	4://区域限定(4:skyRetract)
		CASE phyIdx OF
			0:	lgcIdx := 185;		//sky0r	->	起竖
			1:	lgcIdx := 175;		//sky1r	->	横1
			2:	lgcIdx := 183;		//sky2r	->	纵1
			3:	lgcIdx := 176;		//sky3r	->	横2
			4:	lgcIdx := 177;		//sky4r	->	横3
			5:	lgcIdx := 178;		//sky5r	->	横4
			6:	lgcIdx := 179;		//sky6r	->	横5
			7:	lgcIdx := 184;		//sky7r	->	纵2
			8:	lgcIdx := 180;		//sky8r	->	横6
			9:	lgcIdx := 181;		//sky9r	->	横7
			10:	lgcIdx := 182;		//sky10r->	横8
		END_CASE
END_CASE

END_FUNCTION_BLOCK

// Device/Application/modbus/mdbsNumToIdx
FUNCTION_BLOCK mdbsNumToIdx
VAR_INPUT
	devNo		:WORD;
END_VAR
VAR_OUTPUT
	level		:INT;
	idx			:INT;
END_VAR
VAR
	
END_VAR

IF devNo > 40000 THEN
	CASE devNo OF
		//地轨
		41010:	level := 1;	idx := 1;
		41020:	level := 1;	idx := 3;
		41030:	level := 1;	idx := 4;
		41040:	level := 1;	idx := 5;
		41050:	level := 1;	idx := 6;
		41060:	level := 1;	idx := 8;
		41070:	level := 1;	idx := 9;
		41080:	level := 1;	idx := 10;
		42010:	level := 1;	idx := 2;
		42020:	level := 1;	idx := 7;
		
		51010:	level := 2;	idx := 1;
		51020:	level := 2;	idx := 3;
		51030:	level := 2;	idx := 4;
		51040:	level := 2;	idx := 5;
		51050:	level := 2;	idx := 6;
		51060:	level := 2;	idx := 8;
		51070:	level := 2;	idx := 9;
		51080:	level := 2;	idx := 10;
		52010:	level := 2;	idx := 2;
		52020:	level := 2;	idx := 7;
		53000:	level := 2;	idx := 0;
		53010:	level := 2;	idx := 0;
	END_CASE
END_IF

END_FUNCTION_BLOCK

// Device/Application/modbus/DataReverse
FUNCTION_BLOCK DataReverse
VAR_INPUT
END_VAR
VAR_OUTPUT
END_VAR
VAR
END_VAR

METHOD cmdReverse : TargetDirect
VAR_INPUT
	input		:TargetDirect;
END_VAR
IF input = TargetDirect.extend THEN
	cmdReverse := TargetDirect.retract;
END_IF
IF input = TargetDirect.retract THEN
	cmdReverse := TargetDirect.extend;
END_IF
END_METHOD

END_FUNCTION_BLOCK

// Device/Application/healthydata/TcpUploader
PROGRAM TcpUploader
VAR
	destIp 			:STRING:='172.18.150.31';
	destPort 		:UINT:= 61158;
	tcpConnector	:tcpUpload;
	
	myData 			:ARRAY[1..1024]OF BYTE;
	myDataLen		:__XINT:=21 * 3 + 16;		//总数据长度
	
	init			:BOOL :=TRUE;	
END_VAR



//initialize
IF init THEN
	init := FALSE;
	tcpConnector(InetAddress := destIp,port:= destPort);
END_IF

prepareMetaData();

tcpConnector.send(dataLength := myDataLen, sendBuf := myData);

METHOD prepareMetaData
VAR_INPUT
END_VAR
VAR
	gi				:INT;
	si				:INT;
	
	intTmp			:UINT;	
	pos				:INT;
	byte1			:BYTE;
	byte2			:BYTE;
	plugStat		:BYTE;
END_VAR
//data head (decimal)
myData[1]	:=	83	;
myData[2]	:=	70	;
myData[3]	:=	68	;
myData[4]	:=	84	;

//data length
myData[5]	:=	0	;
myData[6]	:=	63	;

//healthy data
myData[7]	:=	0	;
myData[8]	:=	11	;

//zero
myData[9]	:=	0	;
myData[10]	:=	0	;
myData[11]	:=	0	;
myData[12]	:=	0	;

myData[13]	:=	0	;
myData[14]	:=	0	;
myData[15]	:=	0	;
myData[16]	:=	0	;

//list
pos := 17;
FOR gi := 1 TO 10 DO
	intTmp := REAL_TO_UINT(gDev.grd[gi].sensor.position * 10);
	byte1 := UINT_TO_BYTE(SHR(intTmp, 8)); 
	byte2 := UINT_TO_BYTE(intTmp AND 255); 
	plugStat := INT_TO_BYTE(gDev.grd[gi].state);
	
	myData[pos] := plugStat;
	pos := pos + 1;		
	myData[pos] := byte1;
	pos := pos + 1;
	myData[pos] := byte2;
	pos := pos + 1;
END_FOR
FOR si := 0 TO 10 DO
	intTmp := REAL_TO_UINT(gDev.sky[si].sensor.position * 10);
	byte1 := UINT_TO_BYTE(SHR(intTmp, 8)); 
	byte2 := UINT_TO_BYTE(intTmp AND 255); 
	plugStat := INT_TO_BYTE(gDev.sky[si].state);
	
	myData[pos] := plugStat;
	pos := pos + 1;		
	myData[pos] := byte1;
	pos := pos + 1;
	myData[pos] := byte2;
	pos := pos + 1;
END_FOR
END_METHOD

END_PROGRAM

// Device/Application/basefun/tcpUpload
FUNCTION_BLOCK tcpUpload
VAR_INPUT
	InetAddress		:STRING;
	port			:UINT;
END_VAR
VAR_OUTPUT
END_VAR
VAR
	tcpConnector	:TCP.Connector;
	tcpStream		:TCP.Stream;
	pointerStream	:POINTER TO TCP.Stream;


	tcpState		:UINT:=0;
	tcpCount		:UINT:=0;
	
	netState		:INT;


END_VAR

METHOD send
VAR_INPUT
	
	dataLength		:__XINT;
	sendBuf 		:ARRAY[1..1024]OF BYTE;
END_VAR
VAR
	sizeData		:__XINT;
END_VAR

tcpCount := tcpCount + 1;

CASE tcpState OF

	0:			//connet server
		tcpConnector.Connect(sIPAddress:= InetAddress,uiPort:= port,pStream => pointerStream);
		IF pointerStream<>0 THEN
			tcpState :=1;
		ELSE
			tcpState :=2;
		END_IF
		
	1:			
		netState := pointerStream^.Send(ADR(sendBuf),dataLength,diSent=>sizeData);			
		IF netState <> 0 THEN
			tcpState := 2;	
		END_IF
		
		
	2:		 	//断开连接
	    tcpConnector.Disconnect();
		tcpState := 0;

END_CASE
END_METHOD

END_FUNCTION_BLOCK

// Device/Application/healthydata/FileSaver
PROGRAM FileSaver
VAR
	path 			:STRING:='D:/log';
	intervalMs		:INT := 10;		//间隔时间
	
	init			:BOOL:= TRUE;
	gi				:INT;
	si				:INT;	
	cCtrl			:INT;

	sav				:ARRAY[1..2, 0..10] OF fileSave;
	speed			:INT;
	nowCmd			:ARRAY[1..2, 0..10] OF BOOL;
	canWrite		:ARRAY[1..2, 0..10] OF BOOL;
	nowPosition		:ARRAY[1..2, 0..10] OF INT;
	lastPosition	:ARRAY[1..2, 0..10] OF INT;
	state			:ARRAY[1..2, 0..10] OF INT;
	flag			:ARRAY[1..2, 0..10] OF INT;
END_VAR
VAR CONSTANT
	aOil	:ARRAY [1..7] OF INT :=[9,11,8,8,8,8,23];		
END_VAR

//initialize
IF init THEN
	init := FALSE;
	FOR gi := 1 TO 10 DO
		 sav[1, gi](filePath := path, intervalt := intervalMs);
		 sav[1, gi].createDir(gUI.grd[gi].name);
		 init := FALSE;
	END_FOR
	FOR si := 0 TO 10 DO
		 sav[2, si](filePath := path, intervalt := intervalMs);
		 sav[2, si].createDir(gUI.sky[si].name);
		 init := FALSE;
	END_FOR
END_IF

//detect and record ground and sky
FOR gi := 1 TO 10 DO
	 nowCmd[1, gi] := gUI.grd[gi].btnExtend OR gUI.grd[gi].btnRetract;
	 IF nowCmd[1, gi] THEN
		 IF flag[1, gi] = 0 THEN
			 sav[1, gi].new(devName := gUI.grd[gi].name);
			 flag[1, gi] := 1;
		 END_IF
		 //prepare data
		 getGrdData();
		 //write
		 sav[1, gi].write(positionInt := nowPosition[1, gi],speedInt := speed,
			 				 stateInt := state[1, gi]);
	 ELSE
		 IF flag[1, gi] = 1 THEN
			 sav[1, gi].write(positionInt := nowPosition[1, gi],speedInt := speed,
				 				 stateInt := state[1, gi]);
			 sav[1, gi].close();
			 flag[1, gi] := 0;
		 END_IF
	 END_IF
END_FOR


FOR si := 0 TO 10 DO
	 nowCmd[2, si] := gUI.sky[si].btnExtend OR gUI.sky[si].btnRetract;
	 IF nowCmd[2, si] THEN
		 IF flag[2, si] = 0 THEN
			 sav[2, si].new(devName := gUI.sky[si].name);
			 flag[2, si] := 1;
		 END_IF
		 //prepare data
		 getSkyData();
		 //write
		 sav[2, si].write(positionInt := nowPosition[2, si],speedInt := speed,
			 				 stateInt := state[2, si]);
	 ELSE
		 IF flag[2, si] = 1 THEN
			 sav[2, si].write(positionInt := nowPosition[2, si],speedInt := speed,
				 				 stateInt := state[2, si]);
			 sav[2, si].close();
			 flag[2, si] := 0;
		 END_IF
	 END_IF
END_FOR

ACTION getSkyData:
//进制转换 到0.01mm
lastPosition[2, si] := nowPosition[2, si];
nowPosition[2, si] := REAL_TO_INT(10 * gDev.sky[si].sensor.position);

speed := REAL_TO_INT(gDev.sky[si].sensor.speed);


state[2, si] := gDev.sky[si].state;
END_ACTION

ACTION getGrdData:
//进制转换 到0.01mm
lastPosition[1, gi] := nowPosition[1, gi];
nowPosition[1, gi] := REAL_TO_INT(10 * gDev.grd[gi].sensor.position);

speed := REAL_TO_INT(gDev.grd[gi].sensor.speed);


state[1, gi] := gDev.grd[gi].state;
END_ACTION

END_PROGRAM

// Device/Application/basefun/fileSave
FUNCTION_BLOCK fileSave
VAR_INPUT
	filePath 	:STRING;
	intervalt	:INT;
END_VAR
VAR
	lineCount	: INT;
	fileHandle  : DWORD;
	fileName	: STRING;
END_VAR
VAR_OUTPUT
END_VAR

METHOD new

	
VAR_INPUT
	devName		: STRING ;

END_VAR
VAR
	
	fileHandle0 : DWORD;
	datetime	: DATE_AND_TIME;
	UdIntms 	: UDINT;
	UdMsOffset  : UDINT;
	DTimer_Str  : STRING;
	uiYear 		: UINT; 
    uiMonth 	: UINT; 
    uiDay 		: UINT; 
    uiHour 		: UINT; 
    uiMinute 	: UINT; 
    uiSecond 	: UINT;	
	uiMsSecond	: UINT;



	 S_Time64		:  SysTime64;
	 STT			:  CurTimeEx;
	 S_Time			:  SystemTimeDate;
	 Time_Str		:  STRING;
	F_err		: DWORD;
	F_HANDL		: DWORD;

END_VAR

	STT(SystemTime:= S_Time64, TimeDate:= S_Time);
	Time_Str :='';
	Time_Str := concat(Time_Str,UINT_TO_STRING(S_Time.Year));
	Time_Str := concat(Time_Str,'-');
	Time_Str := concat(Time_Str,UINT_TO_STRING(S_Time.Month));
	Time_Str := concat(Time_Str,'-');
	Time_Str := concat(Time_Str,UINT_TO_STRING(S_Time.Day));
	Time_Str := concat(Time_Str,'_');
	Time_Str := concat(Time_Str,UINT_TO_STRING(S_Time.Hour));
	Time_Str := concat(Time_Str,'-');
	Time_Str := concat(Time_Str,UINT_TO_STRING(S_Time.Minute));
	Time_Str := concat(Time_Str,'-');
	Time_Str := concat(Time_Str,UINT_TO_STRING(S_Time.Second));
	Time_Str := concat(Time_Str,'_');
	Time_Str := concat(Time_Str,UINT_TO_STRING(S_Time.Milliseconds));

	fileName := FilePath;
	fileName := concat(fileName,'/');
	fileName := concat(fileName,devName);

	
	fileName := concat(fileName,'/');
	fileName := concat(fileName,devName);
	fileName := concat(fileName,'-');
	fileName := concat(fileName,Time_Str);
    fileName := concat(fileName,'.txt');

	fileHandle := SysFileOpen(szFile:= fileName, am:=ACCESS_MODE.AM_WRITE, pResult:= ADR(F_err));
	lineCount := -1;
	//fileHandle := SysFileOpen(szFile:= fileName, am:=ACCESS_MODE.AM_APPEND, pResult:= ADR(F_err));
END_METHOD

METHOD close
VAR_INPUT
END_VAR
IF fileHandle <> 0 THEN
	SysFileClose(hFile := fileHandle);
	fileHandle := 0;
END_IF
END_METHOD

METHOD write
VAR_INPUT

	positionInt 	:INT;
	speedInt 		:INT;
	stateInt		:INT;
	
END_VAR
VAR
	data		: STRING;
	F_err		: DWORD;
	tempInt		: INT;
END_VAR

IF fileHandle <> 0 THEN
	lineCount := lineCount + 1;
	tempInt	:= lineCount * intervalt;
	data := INT_TO_STRING(lineCount);
	data := concat(data,'$T$T');
	data := concat(data, INT_TO_STRING(tempInt));
	IF tempInt < 1000 THEN
		data := concat(data,'$T');
	END_IF
	data := concat(data,'$T$T');
	data := concat(data,INT_TO_STRING(positionInt));
	data := concat(data,'$T');
	data := concat(data,INT_TO_STRING(speedInt));
	data := concat(data,'$T');
	data := concat(data,INT_TO_STRING(stateInt));
	data := concat(data,'$R');
	
	SysFileWrite(hFile:=fileHandle , pbyBuffer:= ADR(data) , ulSize:= DINT_TO_DWORD(SysStrLen(data)) , pResult:= ADR(F_err));		// 写入数据

END_IF
END_METHOD

METHOD createDir
VAR_INPUT
	devName		: STRING ;
END_VAR
VAR
	filePath1	:STRING;
END_VAR
filePath1 := FilePath;
filePath1 := concat(filePath1,'/');
filePath1 := concat(filePath1,devName);
SysDirCreate2(filePath1, TRUE);
END_METHOD

END_FUNCTION_BLOCK

// Device/Application/visualization/baseModule/DevUnit0
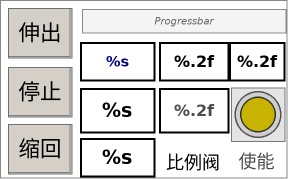
VISUALIZATION DevUnit0  // 288x179
VAR_IN_OUT
	extendButton		: BOOL;
	retractButton		: BOOL;
	stopButton			: BOOL;
	
	percentShow			:REAL;	
	nameShow			:STRING;
	wnameShow			:WSTRING;
	hzname				:WSTRING;
	posShow				:REAL;
	spdShow				:REAL;
	
	pwrEnable			:BOOL;
	pwrPct				:REAL;

END_VAR
    RoundedRectangle (159,88 70x45), "%.2f", text variable: pwrPct
        OnMouseDown: write the text variable via Default, min 0, max 100
    Label (159,149 68x28), "比例阀"
    PushSwitchLed (231,87 54x55), variable: pwrEnable, behaviour: TOGGLE, style: Switch-PushSwitchLed-Yellow
    Label (231,151 51x22), "使能"
    RoundedRectangle (80,42 75x39), "%s", text variable: nameShow
    RoundedRectangle (159,42 70x39), "%.2f", text variable: posShow
    Progressbar (82,9 204x24), variable: percentShow
    Button (8,124 64x50), "缩回"
        toggle retractButton
    Button (8,67 64x50), "停止"
        toggle stopButton
    Button (8,8 64x50), "伸出"
        toggle extendButton
    RoundedRectangle (229,42 56x39), "%.2f", text variable: spdShow
    RoundedRectangle (80,88 75x45), "%s", text variable: wnameShow
    RoundedRectangle (80,138 75x39), "%s", text variable: hzname
END_VISUALIZATION

// Device/Application/visualization/baseModule/grd
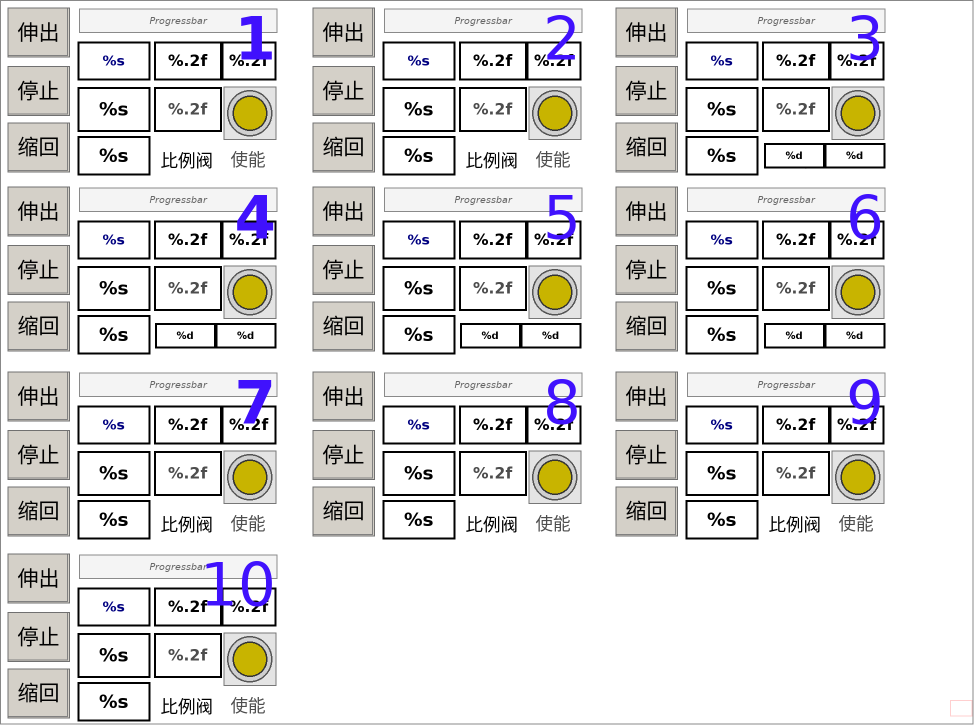
VISUALIZATION grd  // 974x725
    Frame (0,0 279x177), "1"
        shows DevUnit0(extendButton := gUI.grd[1].btnExtend, retractButton := gUI.grd[1].btnRetract, stopButton := gUI.grd[1].btnStop, percentShow := gUI.grd[1].extendPercent, nameShow := gUI.grd[1].name, wnameShow := gUI.grd[1].wname, hzname := gUI.grd[1].hzname, posShow := gUI.grd[1].postion, spdShow := gUI.grd[1].speed, pwrEnable := gUI.grd[1].pwrEnable, pwrPct := gUI.grd[1].pwrPercent)
    Frame (305,0 279x177), "2"
        shows DevUnit0(extendButton := gUI.grd[2].btnExtend, retractButton := gUI.grd[2].btnRetract, stopButton := gUI.grd[2].btnStop, percentShow := gUI.grd[2].extendPercent, nameShow := gUI.grd[2].name, wnameShow := gUI.grd[2].wname, hzname := gUI.grd[2].hzname, posShow := gUI.grd[2].postion, spdShow := gUI.grd[2].speed, pwrEnable := gUI.grd[2].pwrEnable, pwrPct := gUI.grd[2].pwrPercent)
    Frame (608,0 279x177), "3"
        shows DevUnit0(extendButton := gUI.grd[3].btnExtend, retractButton := gUI.grd[3].btnRetract, stopButton := gUI.grd[3].btnStop, percentShow := gUI.grd[3].extendPercent, nameShow := gUI.grd[3].name, wnameShow := gUI.grd[3].wname, hzname := gUI.grd[3].hzname, posShow := gUI.grd[3].postion, spdShow := gUI.grd[3].speed, pwrEnable := gUI.grd[3].pwrEnable, pwrPct := gUI.grd[3].pwrPercent)
    Frame (0,179 279x177), "4"
        shows DevUnit0(extendButton := gUI.grd[4].btnExtend, retractButton := gUI.grd[4].btnRetract, stopButton := gUI.grd[4].btnStop, percentShow := gUI.grd[4].extendPercent, nameShow := gUI.grd[4].name, wnameShow := gUI.grd[4].wname, hzname := gUI.grd[4].hzname, posShow := gUI.grd[4].postion, spdShow := gUI.grd[4].speed, pwrEnable := gUI.grd[4].pwrEnable, pwrPct := gUI.grd[4].pwrPercent)
    Frame (305,179 279x177), "5"
        shows DevUnit0(extendButton := gUI.grd[5].btnExtend, retractButton := gUI.grd[5].btnRetract, stopButton := gUI.grd[5].btnStop, percentShow := gUI.grd[5].extendPercent, nameShow := gUI.grd[5].name, wnameShow := gUI.grd[5].wname, hzname := gUI.grd[5].hzname, posShow := gUI.grd[5].postion, spdShow := gUI.grd[5].speed, pwrEnable := gUI.grd[5].pwrEnable, pwrPct := gUI.grd[5].pwrPercent)
    Frame (608,179 279x177), "6"
        shows DevUnit0(extendButton := gUI.grd[6].btnExtend, retractButton := gUI.grd[6].btnRetract, stopButton := gUI.grd[6].btnStop, percentShow := gUI.grd[6].extendPercent, nameShow := gUI.grd[6].name, wnameShow := gUI.grd[6].wname, hzname := gUI.grd[6].hzname, posShow := gUI.grd[6].postion, spdShow := gUI.grd[6].speed, pwrEnable := gUI.grd[6].pwrEnable, pwrPct := gUI.grd[6].pwrPercent)
    Frame (0,364 279x177), "7"
        shows DevUnit0(extendButton := gUI.grd[7].btnExtend, retractButton := gUI.grd[7].btnRetract, stopButton := gUI.grd[7].btnStop, percentShow := gUI.grd[7].extendPercent, nameShow := gUI.grd[7].name, wnameShow := gUI.grd[7].wname, hzname := gUI.grd[7].hzname, posShow := gUI.grd[7].postion, spdShow := gUI.grd[7].speed, pwrEnable := gUI.grd[7].pwrEnable, pwrPct := gUI.grd[7].pwrPercent)
    Frame (305,364 279x177), "8"
        shows DevUnit0(extendButton := gUI.grd[8].btnExtend, retractButton := gUI.grd[8].btnRetract, stopButton := gUI.grd[8].btnStop, percentShow := gUI.grd[8].extendPercent, nameShow := gUI.grd[8].name, wnameShow := gUI.grd[8].wname, hzname := gUI.grd[8].hzname, posShow := gUI.grd[8].postion, spdShow := gUI.grd[8].speed, pwrEnable := gUI.grd[8].pwrEnable, pwrPct := gUI.grd[8].pwrPercent)
    Frame (608,364 279x177), "9"
        shows DevUnit0(extendButton := gUI.grd[9].btnExtend, retractButton := gUI.grd[9].btnRetract, stopButton := gUI.grd[9].btnStop, percentShow := gUI.grd[9].extendPercent, nameShow := gUI.grd[9].name, wnameShow := gUI.grd[9].wname, hzname := gUI.grd[9].hzname, posShow := gUI.grd[9].postion, spdShow := gUI.grd[9].speed, pwrEnable := gUI.grd[9].pwrEnable, pwrPct := gUI.grd[9].pwrPercent)
    Frame (0,546 279x177), "10"
        shows DevUnit0(extendButton := gUI.grd[10].btnExtend, retractButton := gUI.grd[10].btnRetract, stopButton := gUI.grd[10].btnStop, percentShow := gUI.grd[10].extendPercent, nameShow := gUI.grd[10].name, wnameShow := gUI.grd[10].wname, hzname := gUI.grd[10].hzname, posShow := gUI.grd[10].postion, spdShow := gUI.grd[10].speed, pwrEnable := gUI.grd[10].pwrEnable, pwrPct := gUI.grd[10].pwrPercent)
    Frame (764,143 123x27)
        shows currentUnit(Ixt := gDev.grd[3].current[1], Irt := gDev.grd[3].current[2])
    Frame (155,323 123x27)
        shows currentUnit(Ixt := gDev.grd[4].current[1], Irt := gDev.grd[4].current[2])
    Frame (460,323 123x27)
        shows currentUnit(Ixt := gDev.grd[5].current[1], Irt := gDev.grd[5].current[2])
    Frame (764,323 123x27)
        shows currentUnit(Ixt := gDev.grd[6].current[1], Irt := gDev.grd[6].current[2])
    Rectangle (950,700 22x16)
END_VISUALIZATION

// Device/Application/visualization/baseModule/setting
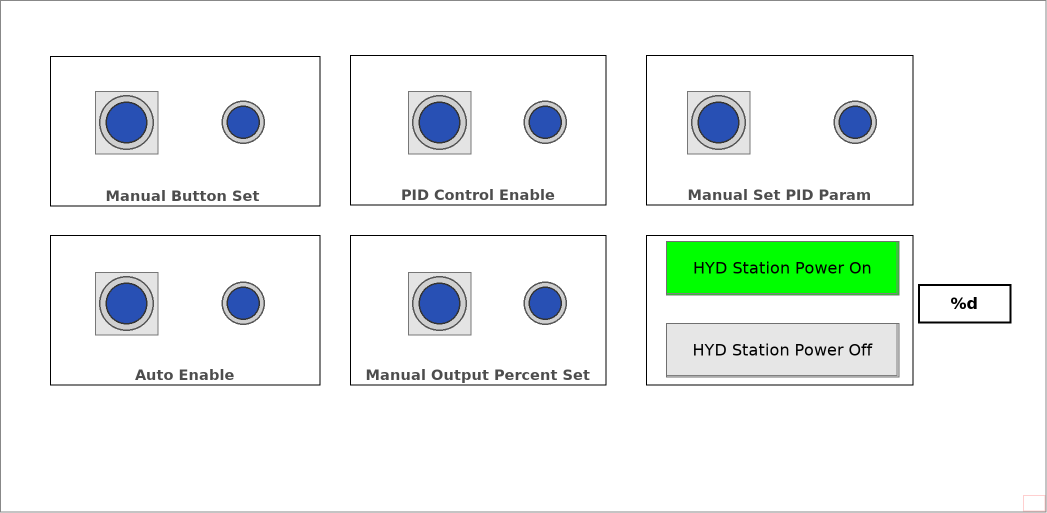
VISUALIZATION setting  // 1047x513
    Rectangle (646,235 267x150)
    Rectangle (50,56 270x150), "Manual Button Set"
    Lamp1 (218,97 50x50), variable: gUI.mode.manualButtonSet, style: Lamp-Lamp1-Blue
    PushSwitchLed (95,90 63x65), variable: gUI.mode.manualButtonSet, behaviour: TOGGLE, style: Switch-PushSwitchLed-Blue
    Rectangle (350,55 256x150), "PID Control Enable"
    Lamp1 (520,97 50x50), variable: gUI.mode.usePID, style: Lamp-Lamp1-Blue
    PushSwitchLed (408,90 63x65), variable: gUI.mode.usePID, behaviour: TOGGLE, style: Switch-PushSwitchLed-Blue
    Rectangle (1023,495 22x16)
    Rectangle (50,235 270x150), "Auto Enable"
    Lamp1 (218,278 50x50), variable: gUI.mode.autoEnable, style: Lamp-Lamp1-Blue
    PushSwitchLed (95,271 63x65), variable: gUI.mode.autoEnable, behaviour: TOGGLE, style: Switch-PushSwitchLed-Blue
    Rectangle (350,235 256x150), "Manual Output Percent Set"
    Lamp1 (520,278 50x50), variable: gUI.mode.manualPercentSet, style: Lamp-Lamp1-Blue
    PushSwitchLed (408,271 63x65), variable: gUI.mode.manualPercentSet, behaviour: TOGGLE, style: Switch-PushSwitchLed-Blue
    Rectangle (646,55 267x150), "Manual Set PID Param"
    Lamp1 (830,97 50x50), variable: gUI.mode.manualSetPid, style: Lamp-Lamp1-Blue
    PushSwitchLed (687,90 63x65), variable: gUI.mode.manualSetPid, behaviour: TOGGLE, style: Switch-PushSwitchLed-Blue
    Button (666,241 233x54), "HYD Station Power On"
        tap gUI.mode.hydPowerOn
    Button (666,323 233x54), "HYD Station Power Off"
        tap gUI.mode.hydPowerOff
    RoundedRectangle (918,284 93x39), "%d", text variable: gModbus.srv.response.data[309]
END_VISUALIZATION

// Device/Application/main
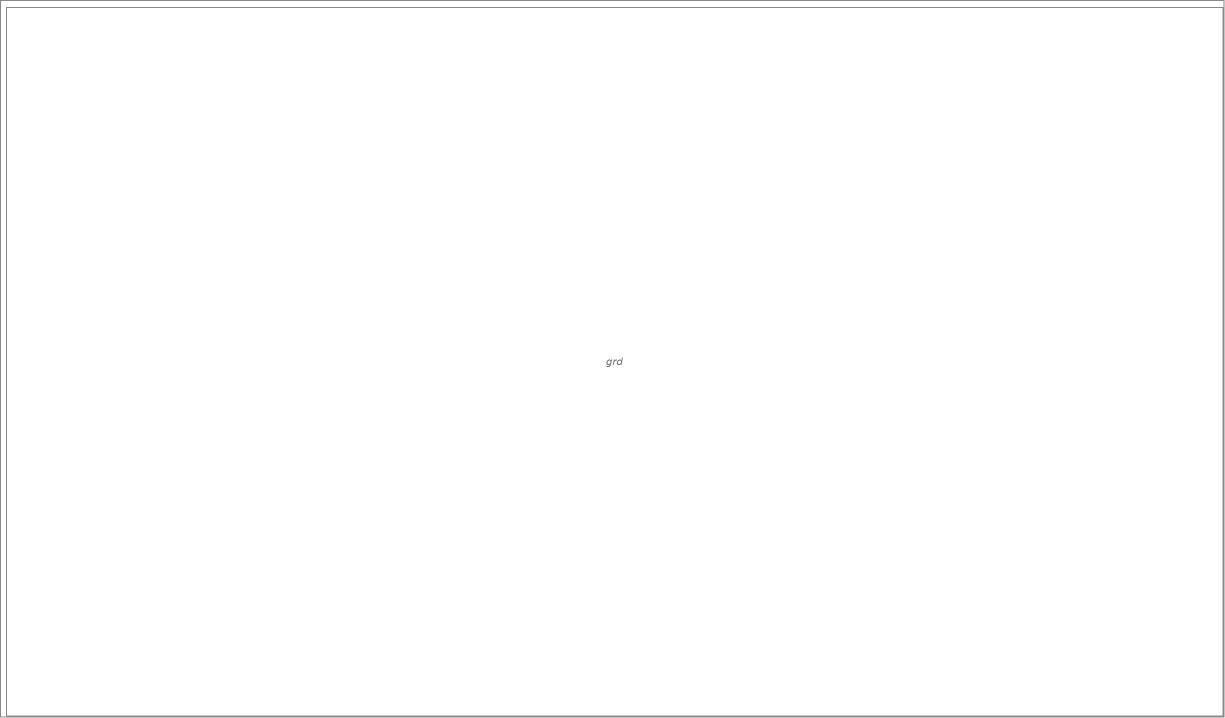
VISUALIZATION main  // 1225x718
    TabControl (6,7 1217x709)
        shows grd()
        shows sky()
        shows testPID()
        shows setting()
        [0]: ImageId=__VisualizationStyle.Element-Switch-PushSwitch-Green-On
        [1]: ImageId=__VisualizationStyle.Element-Switch-PushSwitch-Blue-On
        [2]: ImageId=__VisualizationStyle.Element-Switch-RotarySwitch-Blue-RightUp
        [3]: ImageId=__VisualizationStyle.Element-Switch-PushSwitch-Blue-On
END_VISUALIZATION

// Device/Application/visualization/baseModule/sky
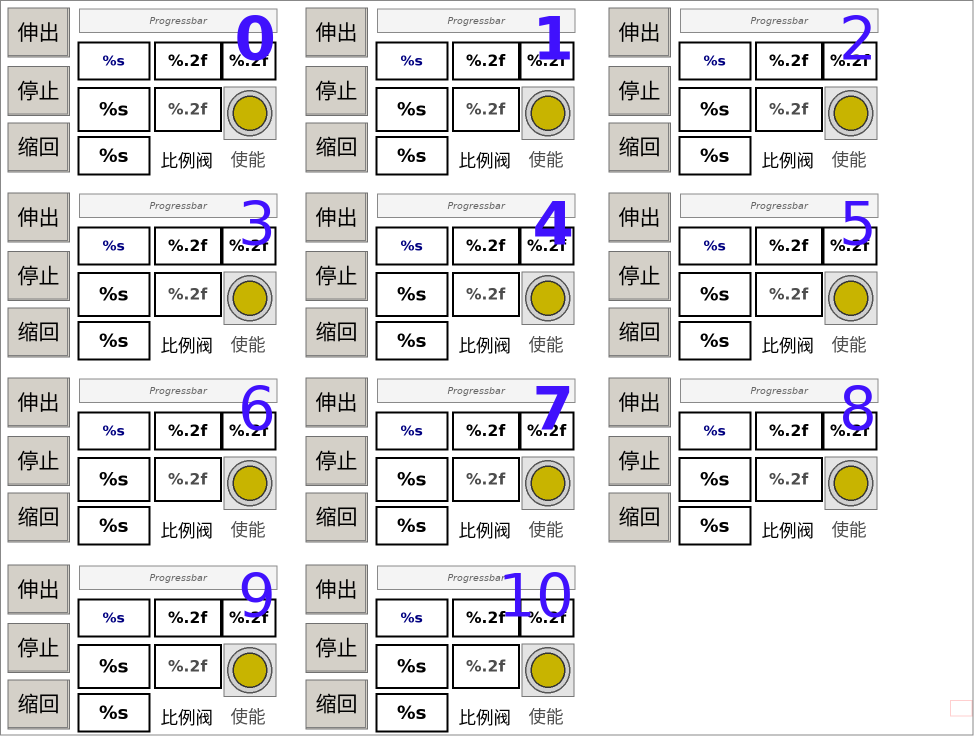
VISUALIZATION sky  // 974x736
    Frame (0,185 279x177), "3"
        shows DevUnit0(extendButton := gUI.sky[3].btnExtend, retractButton := gUI.sky[3].btnRetract, stopButton := gUI.sky[3].btnStop, percentShow := gUI.sky[3].extendPercent, nameShow := gUI.sky[3].name, wnameShow := gUI.sky[3].wname, hzname := gUI.sky[3].hzname, posShow := gUI.sky[3].postion, spdShow := gUI.sky[3].speed, pwrEnable := gUI.sky[3].pwrEnable, pwrPct := gUI.sky[3].pwrPercent)
    Frame (298,185 279x177), "4"
        shows DevUnit0(extendButton := gUI.sky[4].btnExtend, retractButton := gUI.sky[4].btnRetract, stopButton := gUI.sky[4].btnStop, percentShow := gUI.sky[4].extendPercent, nameShow := gUI.sky[4].name, wnameShow := gUI.sky[4].wname, hzname := gUI.sky[4].hzname, posShow := gUI.sky[4].postion, spdShow := gUI.sky[4].speed, pwrEnable := gUI.sky[4].pwrEnable, pwrPct := gUI.sky[4].pwrPercent)
    Frame (601,185 279x177), "5"
        shows DevUnit0(extendButton := gUI.sky[5].btnExtend, retractButton := gUI.sky[5].btnRetract, stopButton := gUI.sky[5].btnStop, percentShow := gUI.sky[5].extendPercent, nameShow := gUI.sky[5].name, wnameShow := gUI.sky[5].wname, hzname := gUI.sky[5].hzname, posShow := gUI.sky[5].postion, spdShow := gUI.sky[5].speed, pwrEnable := gUI.sky[5].pwrEnable, pwrPct := gUI.sky[5].pwrPercent)
    Frame (0,370 279x177), "6"
        shows DevUnit0(extendButton := gUI.sky[6].btnExtend, retractButton := gUI.sky[6].btnRetract, stopButton := gUI.sky[6].btnStop, percentShow := gUI.sky[6].extendPercent, nameShow := gUI.sky[6].name, wnameShow := gUI.sky[6].wname, hzname := gUI.sky[6].hzname, posShow := gUI.sky[6].postion, spdShow := gUI.sky[6].speed, pwrEnable := gUI.sky[6].pwrEnable, pwrPct := gUI.sky[6].pwrPercent)
    Frame (298,370 279x177), "7"
        shows DevUnit0(extendButton := gUI.sky[7].btnExtend, retractButton := gUI.sky[7].btnRetract, stopButton := gUI.sky[7].btnStop, percentShow := gUI.sky[7].extendPercent, nameShow := gUI.sky[7].name, wnameShow := gUI.sky[7].wname, hzname := gUI.sky[7].hzname, posShow := gUI.sky[7].postion, spdShow := gUI.sky[7].speed, pwrEnable := gUI.sky[7].pwrEnable, pwrPct := gUI.sky[7].pwrPercent)
    Frame (601,370 279x177), "8"
        shows DevUnit0(extendButton := gUI.sky[8].btnExtend, retractButton := gUI.sky[8].btnRetract, stopButton := gUI.sky[8].btnStop, percentShow := gUI.sky[8].extendPercent, nameShow := gUI.sky[8].name, wnameShow := gUI.sky[8].wname, hzname := gUI.sky[8].hzname, posShow := gUI.sky[8].postion, spdShow := gUI.sky[8].speed, pwrEnable := gUI.sky[8].pwrEnable, pwrPct := gUI.sky[8].pwrPercent)
    Frame (0,557 279x177), "9"
        shows DevUnit0(extendButton := gUI.sky[9].btnExtend, retractButton := gUI.sky[9].btnRetract, stopButton := gUI.sky[9].btnStop, percentShow := gUI.sky[9].extendPercent, nameShow := gUI.sky[9].name, wnameShow := gUI.sky[9].wname, hzname := gUI.sky[9].hzname, posShow := gUI.sky[9].postion, spdShow := gUI.sky[9].speed, pwrEnable := gUI.sky[9].pwrEnable, pwrPct := gUI.sky[9].pwrPercent)
    Frame (298,557 279x177), "10"
        shows DevUnit0(extendButton := gUI.sky[10].btnExtend, retractButton := gUI.sky[10].btnRetract, stopButton := gUI.sky[10].btnStop, percentShow := gUI.sky[10].extendPercent, nameShow := gUI.sky[10].name, wnameShow := gUI.sky[10].wname, hzname := gUI.sky[10].hzname, posShow := gUI.sky[10].postion, spdShow := gUI.sky[10].speed, pwrEnable := gUI.sky[10].pwrEnable, pwrPct := gUI.sky[10].pwrPercent)
    Frame (298,0 279x177), "1"
        shows DevUnit0(extendButton := gUI.sky[1].btnExtend, retractButton := gUI.sky[1].btnRetract, stopButton := gUI.sky[1].btnStop, percentShow := gUI.sky[1].extendPercent, nameShow := gUI.sky[1].name, wnameShow := gUI.sky[1].wname, hzname := gUI.sky[1].hzname, posShow := gUI.sky[1].postion, spdShow := gUI.sky[1].speed, pwrEnable := gUI.sky[1].pwrEnable, pwrPct := gUI.sky[1].pwrPercent)
    Frame (601,0 279x177), "2"
        shows DevUnit0(extendButton := gUI.sky[2].btnExtend, retractButton := gUI.sky[2].btnRetract, stopButton := gUI.sky[2].btnStop, percentShow := gUI.sky[2].extendPercent, nameShow := gUI.sky[2].name, wnameShow := gUI.sky[2].wname, hzname := gUI.sky[2].hzname, posShow := gUI.sky[2].postion, spdShow := gUI.sky[2].speed, pwrEnable := gUI.sky[2].pwrEnable, pwrPct := gUI.sky[2].pwrPercent)
    Frame (0,0 279x177), "0"
        shows DevUnit0(extendButton := gUI.sky[0].btnExtend, retractButton := gUI.sky[0].btnRetract, stopButton := gUI.sky[0].btnStop, percentShow := gUI.sky[0].extendPercent, nameShow := gUI.sky[0].name, wnameShow := gUI.sky[0].wname, hzname := gUI.sky[0].hzname, posShow := gUI.sky[0].postion, spdShow := gUI.sky[0].speed, pwrEnable := gUI.sky[0].pwrEnable, pwrPct := gUI.sky[0].pwrPercent)
    Rectangle (950,700 22x16)
END_VISUALIZATION

// Device/Application/visualization/baseModule/BasePID
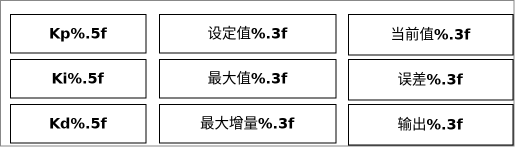
VISUALIZATION BasePID  // 515x147
VAR_IN_OUT
	pid_Kp			:REAL;
	pid_Ki  		:REAL;
	pid_Kd			:REAL;
	pid_Set_Val		:REAL;
	pid_Max_Val		:REAL;
	pid_Max_Acc		:REAL;
	Pid_Act_Val		:REAL;
	Pid_Out			:REAL;
	Pid_Err			:REAL;

END_VAR
    RoundedRectangle (10,14 136x39), "Kp%.5f", text variable: pid_Kp
        OnMouseDown: write the text variable via Default, min 0
    RoundedRectangle (10,59 136x39), "Ki%.5f", text variable: pid_Ki
        OnMouseDown: write the text variable via Default, min 0
    RoundedRectangle (10,104 136x39), "Kd%.5f", text variable: pid_Kd
        OnMouseDown: write the text variable via Default, min 0
    RoundedRectangle (159,14 177x39), "设定值%.3f", text variable: pid_Set_Val
        OnMouseDown: write the text variable via Default
    RoundedRectangle (159,59 177x39), "最大值%.3f", text variable: pid_Max_Val
        OnMouseDown: write the text variable via Default
    RoundedRectangle (159,104 177x39), "最大增量%.3f", text variable: pid_Max_ACC
        OnMouseDown: write the text variable via Default
    RoundedRectangle (348,14 165x41), "当前值%.3f", text variable: Pid_Act_Val
    RoundedRectangle (348,59 165x41), "误差%.3f", text variable: Pid_Err
    RoundedRectangle (348,104 165x41), "输出%.3f", text variable: Pid_Out
END_VISUALIZATION

// Device/Application/visualization/baseModule/testPID
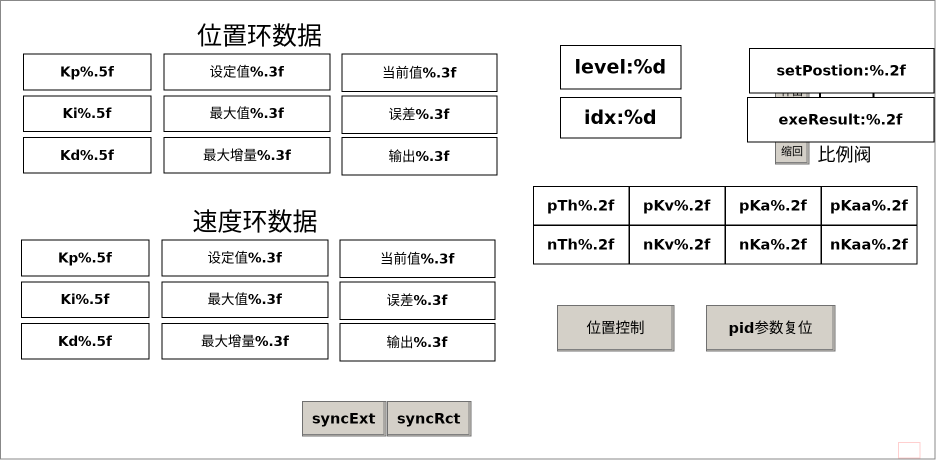
VISUALIZATION testPID  // 936x460
    Frame (14,41 485x136)
        shows BasePID(pid_Kp := gUI.pid.pos.Kp, pid_Ki := gUI.pid.pos.Ki, pid_Kd := gUI.pid.pos.Kd, pid_Set_Val := gUI.pid.pos.Set_Point, pid_Max_Val := gUI.pid.pos.Max_Val, pid_Max_Acc := gUI.pid.pos.Max_ACC, Pid_Act_Val := gUI.pid.pos.Act_Val, Pid_Out := gUI.pid.pos.OUT, Pid_Err := gUI.pid.pos.Err)
    Label (101,15 317x41), "位置环数据"
    Label (107,201 296x41), "速度环数据"
    Frame (12,227 485x136)
        shows BasePID(pid_Kp := gUI.pid.spd.Kp, pid_Ki := gUI.pid.spd.Ki, pid_Kd := gUI.pid.spd.Kd, pid_Set_Val := gUI.pid.spd.Set_Point, pid_Max_Val := gUI.pid.spd.Max_Val, pid_Max_Acc := gUI.pid.spd.Max_ACC, Pid_Act_Val := gUI.pid.spd.Act_Val, Pid_Out := gUI.pid.spd.OUT, Pid_Err := gUI.pid.spd.Err)
    RoundedRectangle (560,97 121x41), "idx:%d", text variable: gUI.pid.idx
        OnMouseDown: write the text variable via Default, min 0, max 10
    RoundedRectangle (560,45 121x44), "level:%d", text variable: gUI.pid.level
        OnMouseDown: write the text variable via Default, min 1, max 2
    Button (557,305 117x46), "位置控制"
        toggle gUI.pid.posBtn
    Rectangle (898,442 22x16)
    Group (775,77 69x56)
        Button (0,62 34x25), "缩回"
            toggle gUI.pid.retractBtn
        Button (0,32 34x25), "停止"
            toggle gUI.pid.stopBtn
        Button (0,2 34x25), "伸出"
            toggle gUI.pid.extendBtn
        RoundedRectangle (44,0 55x24), "%.2f", text variable: gUI.pid.pwrPercent
            OnMouseDown: write the text variable via Default, min 0, max 100
        Label (47,69 45x18), "比例阀"
    Button (706,305 129x46), "pid参数复位"
        tap gUI.pid.rstPidBtn
    Group (533,186 384x78)
        RoundedRectangle (0,0 96x39), "pTh%.2f", text variable: gUI.pid.ff.pstThreshold
            OnMouseDown: write the text variable via Default, min 0
        RoundedRectangle (0,39 96x39), "nTh%.2f", text variable: gUI.pid.ff.negThreshold
            OnMouseDown: write the text variable via Default, min 0
        RoundedRectangle (96,0 96x39), "pKv%.2f", text variable: gUI.pid.ff.pstKv
            OnMouseDown: write the text variable via Default, min 0
        RoundedRectangle (192,0 96x39), "pKa%.2f", text variable: gUI.pid.ff.pstKa
            OnMouseDown: write the text variable via Default, min 0
        RoundedRectangle (288,0 96x39), "pKaa%.2f", text variable: gUI.pid.ff.pstKaa
            OnMouseDown: write the text variable via Default, min 0
        RoundedRectangle (96,39 96x39), "nKv%.2f", text variable: gUI.pid.ff.negKv
            OnMouseDown: write the text variable via Default, min 0
        RoundedRectangle (192,39 96x39), "nKa%.2f", text variable: gUI.pid.ff.negKa
            OnMouseDown: write the text variable via Default, min 0
        RoundedRectangle (288,39 96x39), "nKaa%.2f", text variable: gUI.pid.ff.negKaa
            OnMouseDown: write the text variable via Default, min 0
    RoundedRectangle (747,97 187x45), "exeResult:%.2f", text variable: gUI.pid.executeVal
    RoundedRectangle (749,48 185x45), "setPostion:%.2f", text variable: gUI.pid.devSetPos
    Button (302,401 84x35), "syncExt"
        tap gUI.mode.syncExt
    Button (387,401 84x35), "syncRct"
        tap gUI.mode.syncRct
END_VISUALIZATION

// Device/Application/visualization/baseModule/currentUnit
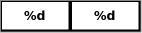
VISUALIZATION currentUnit  // 142x33
VAR_IN_OUT
	Ixt		:	WORD;
	Irt		:	WORD;
END_VAR
    RoundedRectangle (0,0 70x31), "%d", text variable: Ixt
    RoundedRectangle (70,0 70x31), "%d", text variable: Irt
END_VISUALIZATION
